RoboDK station: example.rdk

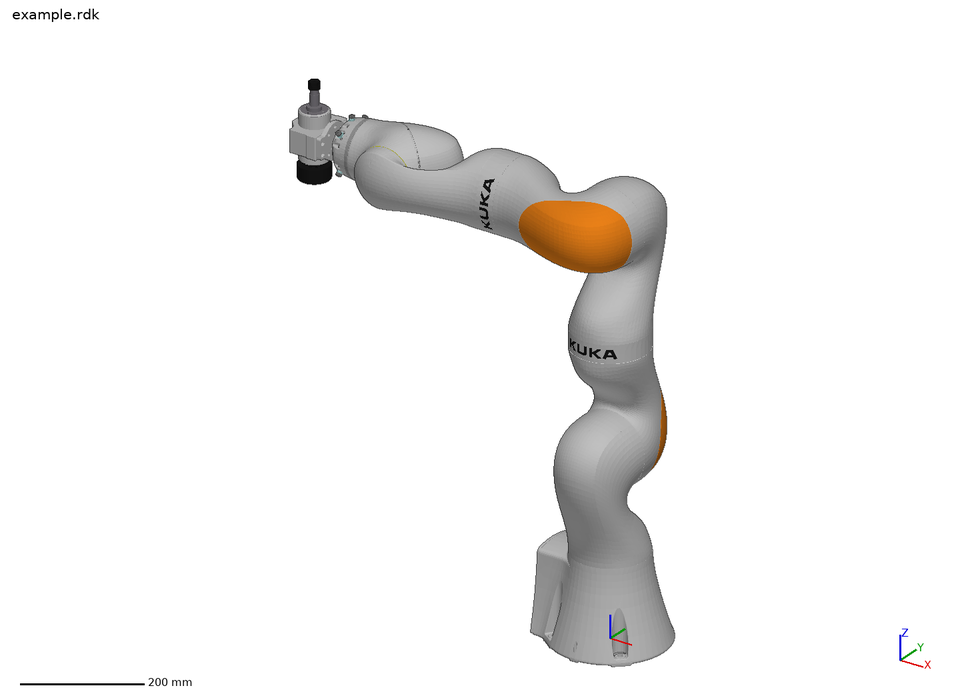
[picture v0: the station drawn from its stored meshes, robots at their saved joint values, targets as dots, program paths as lines]
Station example (saved by RoboDK 5.1.1). Poses are relative to the parent item; angles as X-Y-Z fixed-axis rotations.
  - frame KUKA LBR iiwa 7 R800 Base at (0, 0, 0) mm
    - robot KUKA LBR iiwa 7 R800: 7 axes, payload 7 kg, reach 800 mm, repeatability 0.1 mm, weight 23.9 kg
        modified DH rows (alpha deg, a mm, theta deg, d mm): 0, 0, 0, 340; -90, 0, 0, 0; 90, 0, 0, 400; -90, 0, 0, 0; 90, 0, 0, 400; -90, 0, 0, 0; 90, 0, 0, 130
        joint limits [-170, -120, -170, -120, -170, -120, -175] to [170, 120, 170, 120, 170, 120, 175]; home [0, 0, 0, -90, 0, 0, 0]; saved at [0, 0, 0, -90, 0, 0, 0]
      - tool Spindle, TCP at (118.2, 2.64, 54.29) mm, rotated rx 90 ry 0 rz 90 deg, size 174.1 x 90 x 75.6 mm, geometry from KUKA LBR iiwa 7 R800 Base
  - program HandGuiding (1 instructions, listed below)

--- program HandGuiding (robot KUKA LBR iiwa 7 R800) ---
  Pause 1.0 s
